(* Logix 5000 project; controller PLCbox vendor 1 type 14 code 149 rev 30.11; software revision 30.01; part 4 of 4 *)
(* tags used below, declared in another part *)
   AScaled : REAL;
   BOOL : BOOL[64];
   LocalBOOL : BOOL[64];
   LocalDINT : DINT[20];
   LocDINT : DINT[20];
   MTR1 : BOOL[64];
   Running : BOOL;
   StartPB : BOOL;
   StopButton : BOOL;
   StopPB : DINT;
   TempC : REAL;
   TempF : REAL;
   AnalogInput : REAL[100];
   DINT_Arr1 : DINT[40];
   DINT_Arr2 : DINT[40];
   FaultedT : TIMER;
   HMI_Int_BOOL : BOOL[64];
   Light1_Complete_ONS : BOOL;
   Light1_Green : BOOL;
   Light1_Green_T : TIMER;
   Light1_Red : BOOL;
   Light1_Reset : BOOL;
   Light1_Yellow : BOOL;
   Light1_Yellow_T : TIMER;
   Light2_Complete_ONS : BOOL;
   Light2_Green : BOOL;
   Light2_Green_T : TIMER;
   Light2_Red : BOOL;
   Light2_Reset : BOOL;
   Light2_Yellow : BOOL;
   Light2_Yellow_T : TIMER;
   LightSystem_FLT : BOOL[64];
   LightSystemFaulted : BOOL;
   Local2IData : DINT;
   Local3OData : DINT;
   Local_IN_D : BOOL[256];
   Local_OUT_D : BOOL[256];
   System_Timer : TIMER[100];
   SystemFaultReset : BOOL;
   tagToPi : DINT;
(* ST_Practice, continued *)

ROUTINE _04_MotorStartST   (* structured text *)
   // MTR1[3] - StartPB
   // MTR1[4] - StopPB
   // MTR1[5] - Motor Running
   //MTR1[5] := (MTR1[3] OR MTR1[5]) AND NOT(MTR1[4]);
   IF (MTR1[3] OR MTR1[5]) AND NOT(MTR1[4]) THEN
   MTR1[5] := 1;
   ELSE
   MTR1[5] := 0;
   END_IF;
END_ROUTINE

ROUTINE _05_Practice   (* structured text *)
   
END_ROUTINE

ROUTINE _06_LogicOps   (* structured text *)
   //OR Operator
   LocalBOOL[0] := LocalBOOL[1] OR LocalBOOL[2];
   
   //AND Operator
   LocalBOOL[3] := LocalBOOL[4] AND LocalBOOL[5];
   
   //NOT Operator
   LocalBOOL[6] := NOT(LocalBOOL[7]);
   
   //Motor Starter
   Running [:=] (Running OR StartPB) AND NOT(StopButton);
   
   //GRT, LES, LIM (Not available in ST) -> CMP
   LocalBOOL[8] := 100 + LocalDINT[1] < LocalDINT[0] - 44;
END_ROUTINE

ROUTINE _07_OperatorsFunctions   (* structured text *)
   //Mathematical / Built-In Operators
   LocDINT[0] := LocDINT[1] + 5;
   LocDINT[2] := LocDINT[3] - 4;
   LocDINT[4] := LocDINT[0] * 3;
   LocDINT[5] := 5/LocDINT[1];
   LocDINT[6] := LocDINT[0] ** 3;
   LocDINT[7] := LocDINT[6] MOD 4;
   
   LocDINT[8] := LocDINT[1] + LocDINT[6] / 2 + LocDINT[2];
   
   //Examples
   TempC := (TempF - 32) * 5/9;
   AScaled := AnalogInput[0] / 160 * 3;
END_ROUTINE
END_PROGRAM

PROGRAM StreetLightSystem   (* main routine _01_Main *)
VAR
   HMI_Int_DINT : DINT[100] := ([0] := 10000, [1] := 3000, [2] := 10000, [3] := 3000);
END_VAR

ROUTINE _01_Main   (* ladder *)
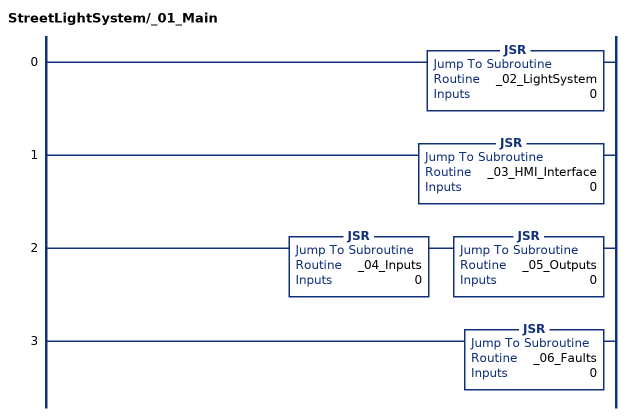
   0: JSR(_02_LightSystem,0);
   1: JSR(_03_HMI_Interface,0);
   2: JSR(_04_Inputs,0)JSR(_05_Outputs,0);
   3: JSR(_06_Faults,0);
END_ROUTINE

ROUTINE _02_LightSystem   (* ladder *)
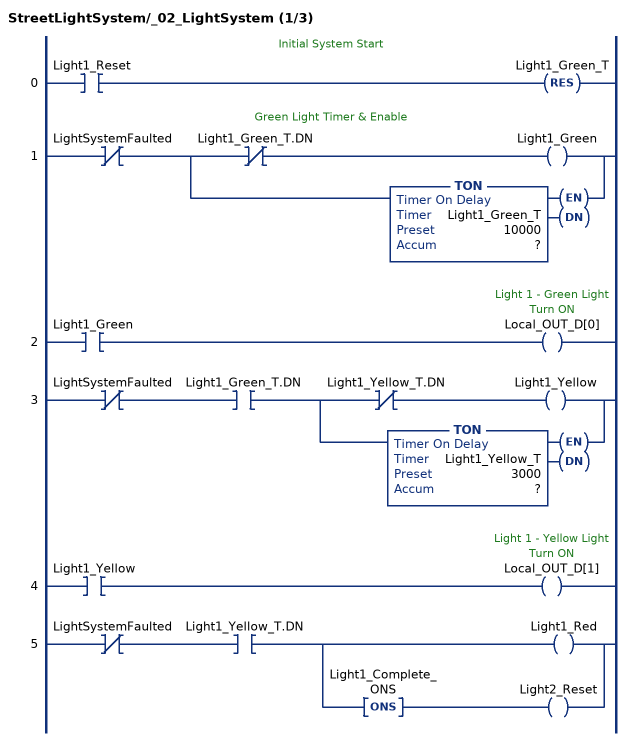
   // Initial System Start
   0: XIC(Light1_Reset)RES(Light1_Green_T);
   // Green Light Timer & Enable
   1: XIO(LightSystemFaulted)[XIO(Light1_Green_T.DN) OTE(Light1_Green) ,TON(Light1_Green_T,?,?) ];
   2: XIC(Light1_Green)OTE(Local_OUT_D[0]);
   3: XIO(LightSystemFaulted)XIC(Light1_Green_T.DN)[XIO(Light1_Yellow_T.DN) OTE(Light1_Yellow) ,TON(Light1_Yellow_T,?,?) ];
   4: XIC(Light1_Yellow)OTE(Local_OUT_D[1]);
   5: XIO(LightSystemFaulted)XIC(Light1_Yellow_T.DN)[OTE(Light1_Red) ,ONS(Light1_Complete_ONS) OTE(Light2_Reset) ];
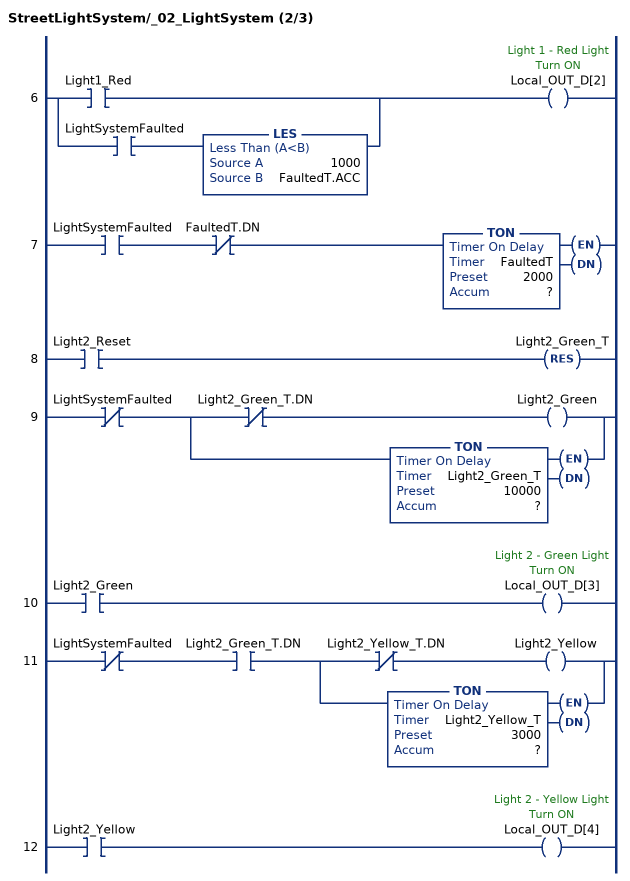
   6: [XIC(Light1_Red) ,XIC(LightSystemFaulted) LES(1000,FaultedT.ACC) ]OTE(Local_OUT_D[2]);
   7: XIC(LightSystemFaulted)XIO(FaultedT.DN)TON(FaultedT,?,?);
   8: XIC(Light2_Reset)RES(Light2_Green_T);
   9: XIO(LightSystemFaulted)[XIO(Light2_Green_T.DN) OTE(Light2_Green) ,TON(Light2_Green_T,?,?) ];
   10: XIC(Light2_Green)OTE(Local_OUT_D[3]);
   11: XIO(LightSystemFaulted)XIC(Light2_Green_T.DN)[XIO(Light2_Yellow_T.DN) OTE(Light2_Yellow) ,TON(Light2_Yellow_T,?,?) ];
   12: XIC(Light2_Yellow)OTE(Local_OUT_D[4]);
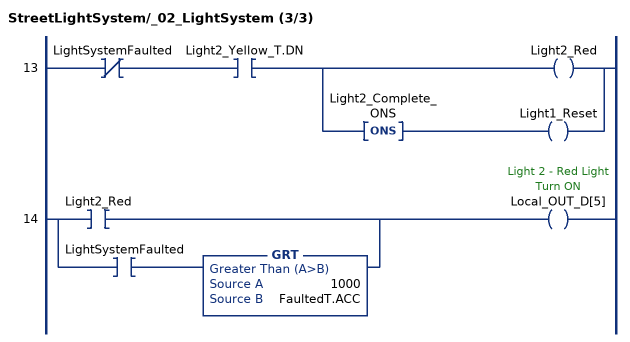
   13: XIO(LightSystemFaulted)XIC(Light2_Yellow_T.DN)[OTE(Light2_Red) ,ONS(Light2_Complete_ONS) OTE(Light1_Reset) ];
   14: [XIC(Light2_Red) ,XIC(LightSystemFaulted) GRT(1000,FaultedT.ACC) ]OTE(Local_OUT_D[5]);
END_ROUTINE

ROUTINE _03_HMI_Interface   (* ladder *)
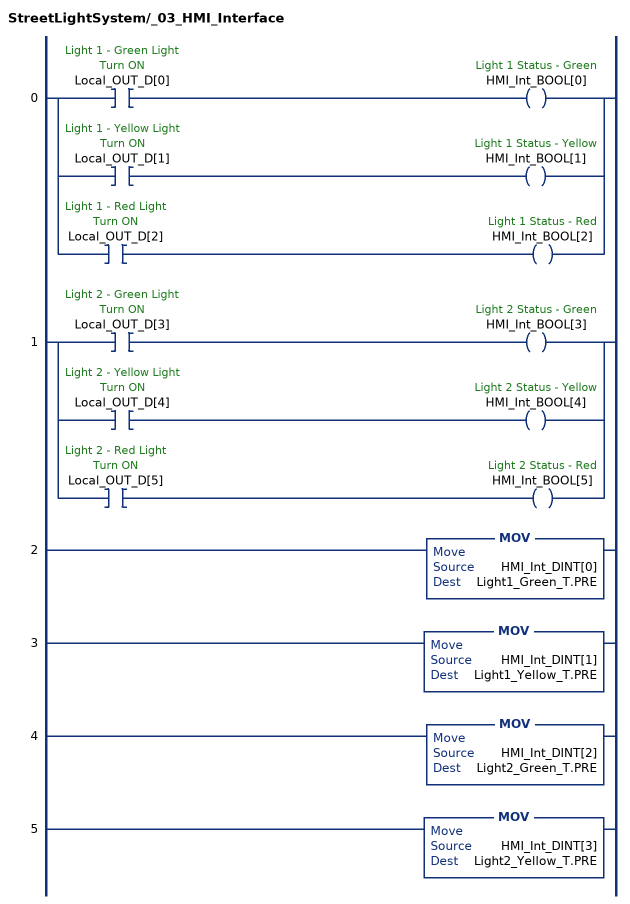
   0: [XIC(Local_OUT_D[0]) OTE(HMI_Int_BOOL[0]) ,XIC(Local_OUT_D[1]) OTE(HMI_Int_BOOL[1]) ,XIC(Local_OUT_D[2]) OTE(HMI_Int_BOOL[2]) ];
   1: [XIC(Local_OUT_D[3]) OTE(HMI_Int_BOOL[3]) ,XIC(Local_OUT_D[4]) OTE(HMI_Int_BOOL[4]) ,XIC(Local_OUT_D[5]) OTE(HMI_Int_BOOL[5]) ];
   2: MOV(HMI_Int_DINT[0],Light1_Green_T.PRE);
   3: MOV(HMI_Int_DINT[1],Light1_Yellow_T.PRE);
   4: MOV(HMI_Int_DINT[2],Light2_Green_T.PRE);
   5: MOV(HMI_Int_DINT[3],Light2_Yellow_T.PRE);
END_ROUTINE

ROUTINE _04_Inputs   (* ladder *)
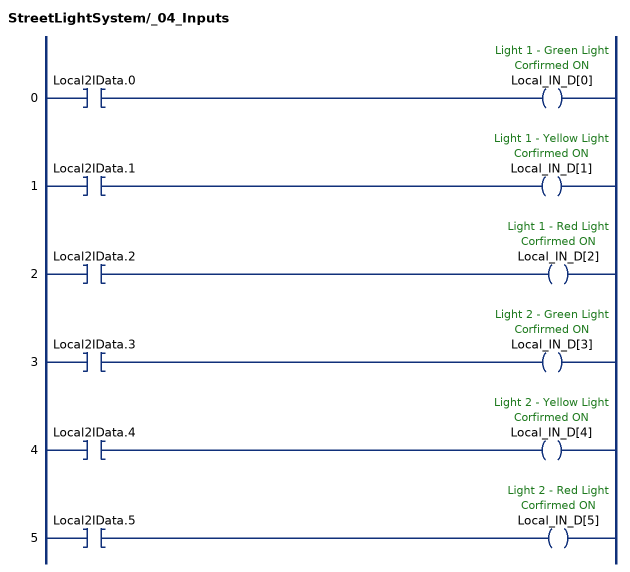
   0: XIC(Local2IData.0)OTE(Local_IN_D[0]);
   1: XIC(Local2IData.1)OTE(Local_IN_D[1]);
   2: XIC(Local2IData.2)OTE(Local_IN_D[2]);
   3: XIC(Local2IData.3)OTE(Local_IN_D[3]);
   4: XIC(Local2IData.4)OTE(Local_IN_D[4]);
   5: XIC(Local2IData.5)OTE(Local_IN_D[5]);
END_ROUTINE

ROUTINE _05_Outputs   (* ladder *)
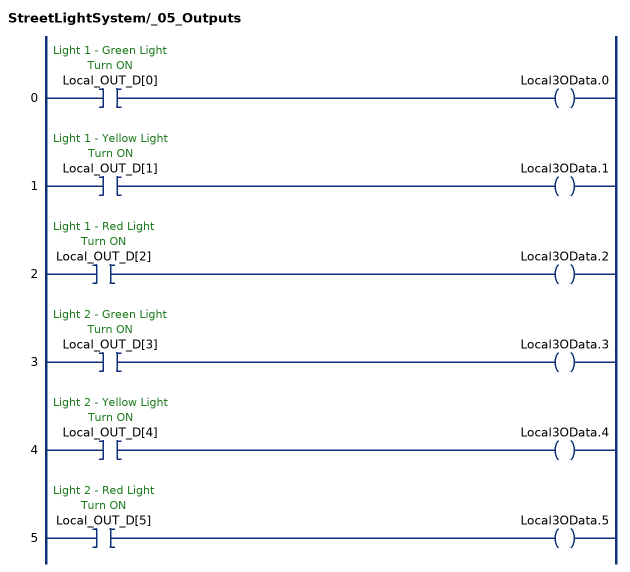
   0: XIC(Local_OUT_D[0])OTE(Local3OData.0);
   1: XIC(Local_OUT_D[1])OTE(Local3OData.1);
   2: XIC(Local_OUT_D[2])OTE(Local3OData.2);
   3: XIC(Local_OUT_D[3])OTE(Local3OData.3);
   4: XIC(Local_OUT_D[4])OTE(Local3OData.4);
   5: XIC(Local_OUT_D[5])OTE(Local3OData.5);
END_ROUTINE

ROUTINE _06_Faults   (* ladder *)
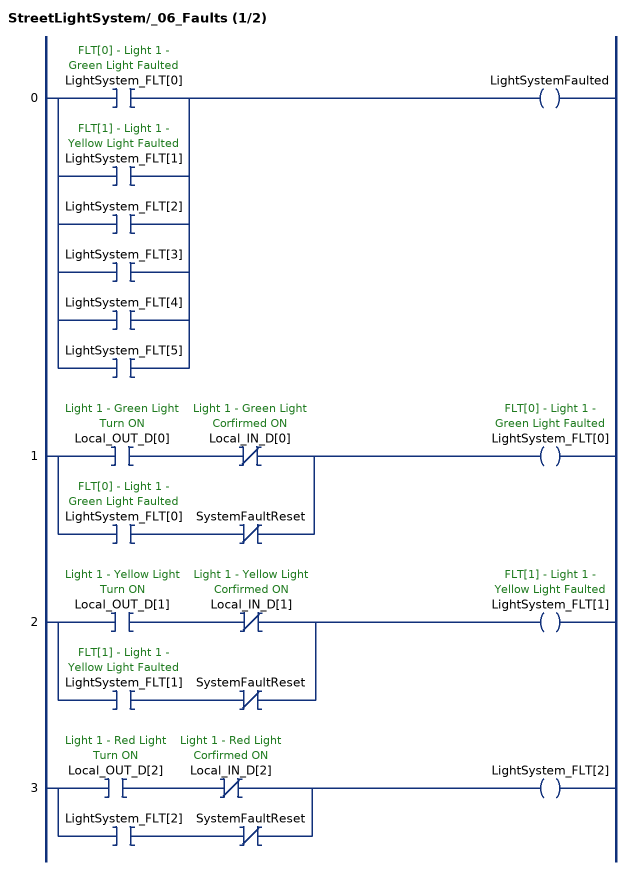
   0: [XIC(LightSystem_FLT[0]) ,XIC(LightSystem_FLT[1]) ,XIC(LightSystem_FLT[2]) ,XIC(LightSystem_FLT[3]) ,XIC(LightSystem_FLT[4]) ,XIC(LightSystem_FLT[5]) ]OTE(LightSystemFaulted);
   1: [XIC(Local_OUT_D[0]) XIO(Local_IN_D[0]) ,XIC(LightSystem_FLT[0]) XIO(SystemFaultReset) ]OTE(LightSystem_FLT[0]);
   2: [XIC(Local_OUT_D[1]) XIO(Local_IN_D[1]) ,XIC(LightSystem_FLT[1]) XIO(SystemFaultReset) ]OTE(LightSystem_FLT[1]);
   3: [XIC(Local_OUT_D[2]) XIO(Local_IN_D[2]) ,XIC(LightSystem_FLT[2]) XIO(SystemFaultReset) ]OTE(LightSystem_FLT[2]);
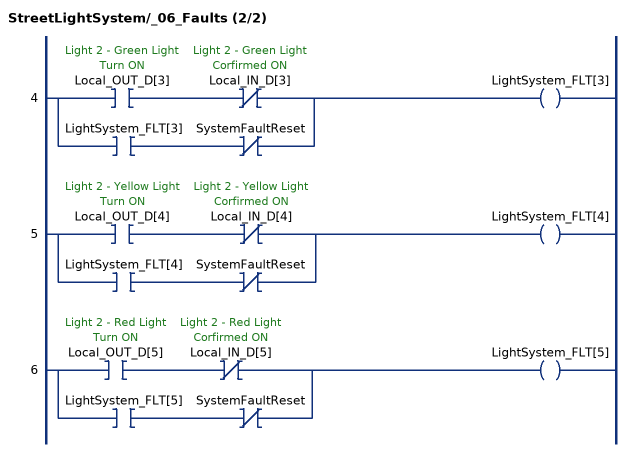
   4: [XIC(Local_OUT_D[3]) XIO(Local_IN_D[3]) ,XIC(LightSystem_FLT[3]) XIO(SystemFaultReset) ]OTE(LightSystem_FLT[3]);
   5: [XIC(Local_OUT_D[4]) XIO(Local_IN_D[4]) ,XIC(LightSystem_FLT[4]) XIO(SystemFaultReset) ]OTE(LightSystem_FLT[4]);
   6: [XIC(Local_OUT_D[5]) XIO(Local_IN_D[5]) ,XIC(LightSystem_FLT[5]) XIO(SystemFaultReset) ]OTE(LightSystem_FLT[5]);
END_ROUTINE
END_PROGRAM

PROGRAM TankFillingChallenge   (* main routine _01_Main *)
VAR
   DischargeStatus : DINT := 1;
   FillingStatus : DINT := 1;
   T_Vlad : BOOL[128];
   TankActualLevel : REAL := 42.792046;
   TankDischargeRate : REAL := 0.5;
   TankEmptyThreshold : REAL := 5.0;
   TankFill : BOOL[128];
        [6]   // TANK FULL
        [7]   // TANK EMPTY
        [2]   // Filling Station RUNNING
        [3]   // START Discharge Station
        [0]   // START Filling Station
        [1]   // STOP Filling Station
        [5]   // Discharge Station RUNNING
        [4]   // STOP Discharge Station
   TankFillRate : REAL := 0.3;
   TankFullThreshold : REAL := 100.0;
   TankOut : BOOL[32];
        [0]   // Filling Station VALVE OPEN
        [1]   // Discharge Station VALVE OPEN
   TankTimers : TIMER[10] := ([0].PRE := 20, [1].PRE := 20);
END_VAR

ROUTINE _01_Main   (* ladder *)
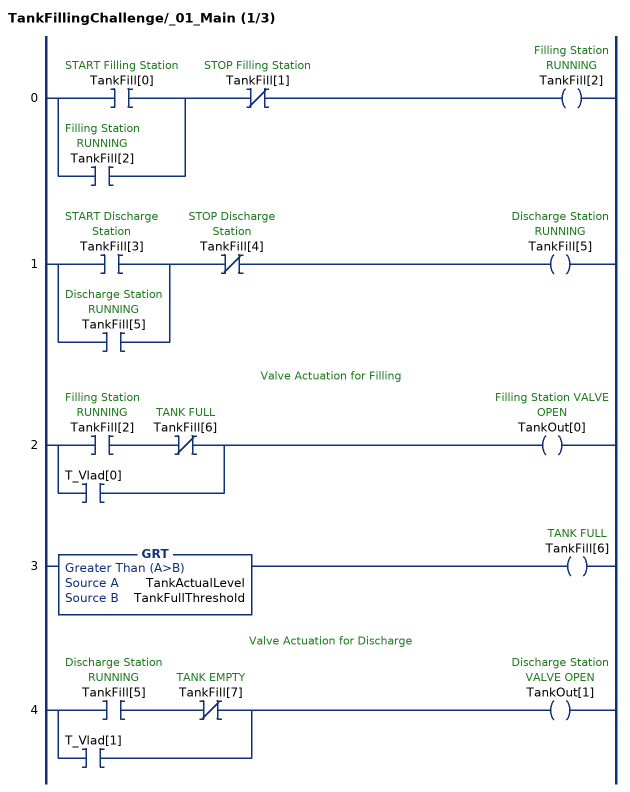
   0: [XIC(TankFill[0]) ,XIC(TankFill[2]) ]XIO(TankFill[1])OTE(TankFill[2]);
   1: [XIC(TankFill[3]) ,XIC(TankFill[5]) ]XIO(TankFill[4])OTE(TankFill[5]);
   // Valve Actuation for Filling
   2: [XIC(TankFill[2]) XIO(TankFill[6]) ,XIC(T_Vlad[0]) ]OTE(TankOut[0]);
   3: GRT(TankActualLevel,TankFullThreshold)OTE(TankFill[6]);
   // Valve Actuation for Discharge
   4: [XIC(TankFill[5]) XIO(TankFill[7]) ,XIC(T_Vlad[1]) ]OTE(TankOut[1]);
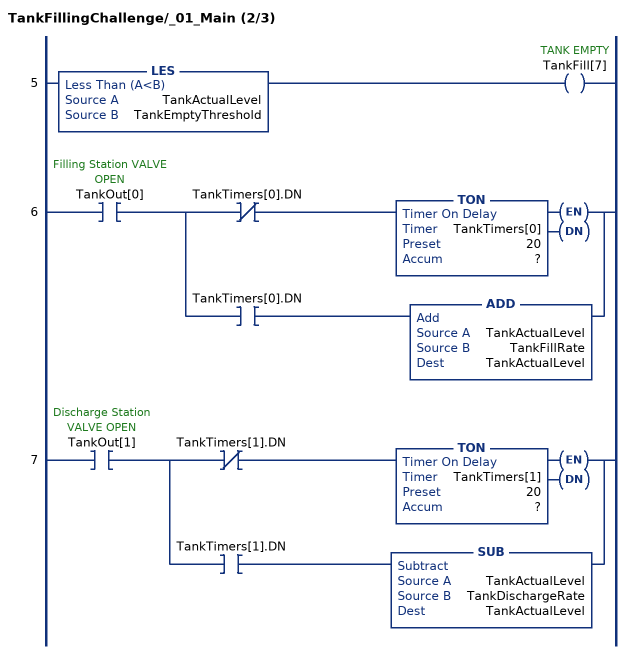
   5: LES(TankActualLevel,TankEmptyThreshold)OTE(TankFill[7]);
   6: XIC(TankOut[0])[XIO(TankTimers[0].DN) TON(TankTimers[0],?,?) ,XIC(TankTimers[0].DN) ADD(TankActualLevel,TankFillRate,TankActualLevel) ];
   7: XIC(TankOut[1])[XIO(TankTimers[1].DN) TON(TankTimers[1],?,?) ,XIC(TankTimers[1].DN) SUB(TankActualLevel,TankDischargeRate,TankActualLevel) ];
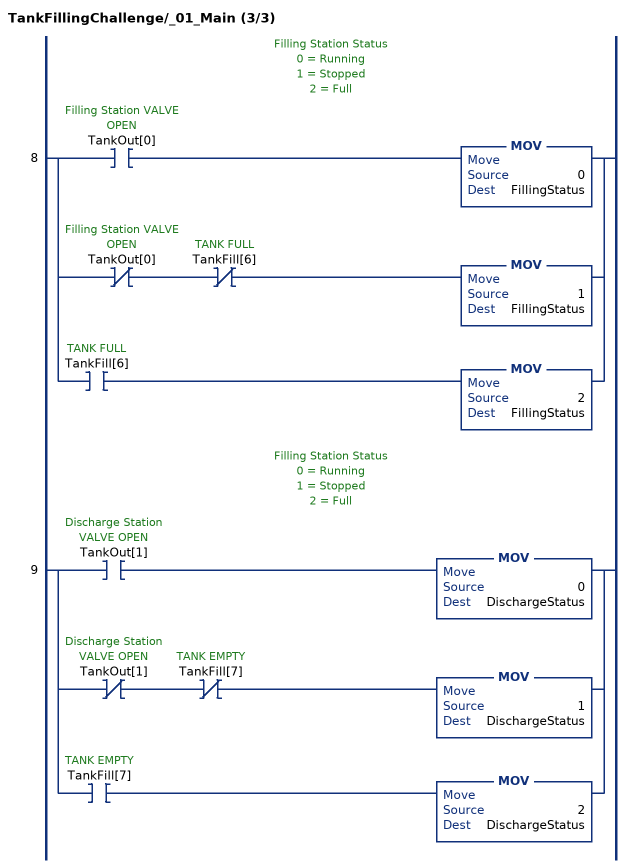
   // Filling Station Status
   // 0 = Running
   // 1 = Stopped
   // 2 = Full
   8: [XIC(TankOut[0]) MOV(0,FillingStatus) ,XIO(TankOut[0]) XIO(TankFill[6]) MOV(1,FillingStatus) ,XIC(TankFill[6]) MOV(2,FillingStatus) ];
   // Filling Station Status
   // 0 = Running
   // 1 = Stopped
   // 2 = Full
   9: [XIC(TankOut[1]) MOV(0,DischargeStatus) ,XIO(TankOut[1]) XIO(TankFill[7]) MOV(1,DischargeStatus) ,XIC(TankFill[7]) MOV(2,DischargeStatus) ];
END_ROUTINE
END_PROGRAM

PROGRAM TestProgram   (* main routine Main *)
VAR
   ALARM : BOOL[256];
   ALARM2 : BOOL[256];
   ALARM_DESC : String20;
   ALARM_DESCR : String20[256] := ([0] := 'Fault 0', [1] := 'Fault 1', [2] := 'Fault 2');
   Condition1 : BOOL := 1;
   Condition10 : BOOL := 1;
   Condition11 : BOOL := 1;
   Condition2 : BOOL;
   Condition3 : BOOL := 1;
   Condition4 : BOOL;
   Condition5 : BOOL := 1;
   Condition6 : BOOL;
   Condition7 : BOOL;
   Condition8 : BOOL := 1;
   Condition9 : BOOL := 1;
   EmptyString : String20;
   Energize : BOOL;
   Energize1 : BOOL := 1;
   FaultDesc : String20 := 'Fault 1';
   FaultDesc2 : String20 := 'Fault 1';
   HMI_BOOL : BOOL[32];
   Index : DINT := 256;
   Motor_1_Start : BOOL;
   Motor_2_Start : BOOL;
   OFFinst : TIMER := (PRE := 500);
   ONinst : TIMER := (PRE := 3000, ACC := 2342, EN := 1, TT := 1);
   PLC_BOOL : BOOL[32];
   Program_Enabled : BOOL;
   Program_Running : BOOL;
   Program_Starting : BOOL;
   RunRoutine : TIMER := (PRE := 500);
   StartProgram : BOOL;
   StartRoutine : TIMER := (PRE := 1000);
   System_Cond : BOOL[256] := ([0] := 1);
        [0]   // Start MOTOR 1
        [2]   // Start MOTOR 2
        [5]   // Boiler at Temp
        [6]   // System Running
        [7]   // System FAULTED
        [1]   // MOTOR 1 At Target Speed
        [8]   // System RESET
        [4]   // Heat Boiler
        [3]   // Motor 2 at Target Speed
   System_INT : INT[10] := ([0] := 456, [1] := 456, [2] := 1);
   System_REAL : REAL[10] := ([0] := 54.0, [1] := 54.0, [2] := 54.0);
   System_STR : STRING[10];
   System_STRING : String20[10];
   SystemFaulted : BOOL := 1;
   SystemFaulted2 : BOOL := 1;
   SystemStart : BOOL;
   SytemReset : BOOL;
   SytemReset2 : BOOL;
   Test1 : DINT := 560647;
   Test2 : INT := -29177;
   TestDINT : DINT;
   TestINT : INT;
END_VAR

ROUTINE _02_MOV_Instruction   (* ladder *)
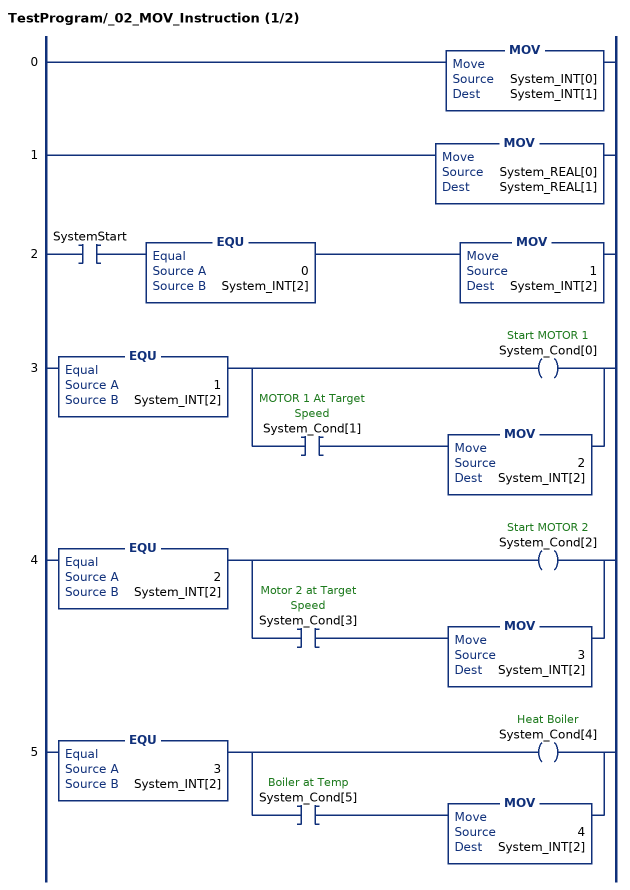
   0: MOV(System_INT[0],System_INT[1]);
   1: MOV(System_REAL[0],System_REAL[1]);
   2: XIC(SystemStart)EQU(0,System_INT[2])MOV(1,System_INT[2]);
   3: EQU(1,System_INT[2])[OTE(System_Cond[0]) ,XIC(System_Cond[1]) MOV(2,System_INT[2]) ];
   4: EQU(2,System_INT[2])[OTE(System_Cond[2]) ,XIC(System_Cond[3]) MOV(3,System_INT[2]) ];
   5: EQU(3,System_INT[2])[OTE(System_Cond[4]) ,XIC(System_Cond[5]) MOV(4,System_INT[2]) ];
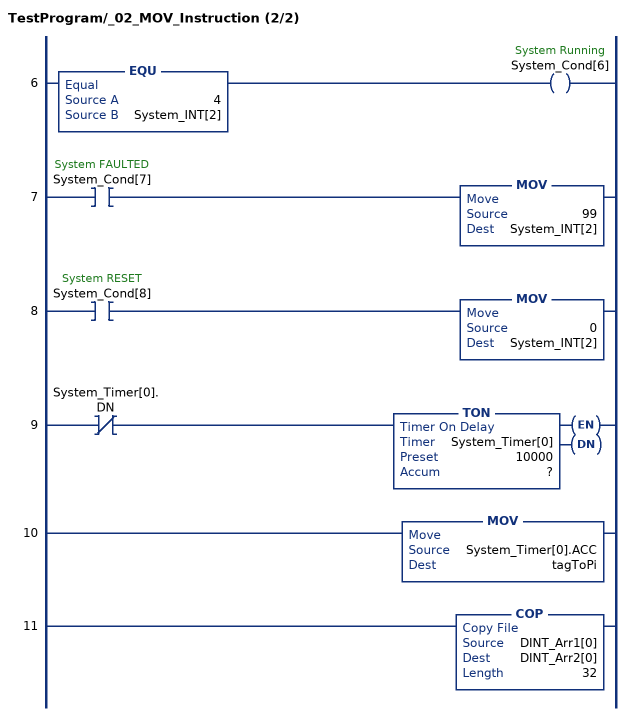
   6: EQU(4,System_INT[2])OTE(System_Cond[6]);
   7: XIC(System_Cond[7])MOV(99,System_INT[2]);
   8: XIC(System_Cond[8])MOV(0,System_INT[2]);
   9: XIO(System_Timer[0].DN)TON(System_Timer[0],?,?);
   10: MOV(System_Timer[0].ACC,tagToPi);
   11: COP(DINT_Arr1[0],DINT_Arr2[0],32);
END_ROUTINE

ROUTINE _03_HMI   (* ladder *)
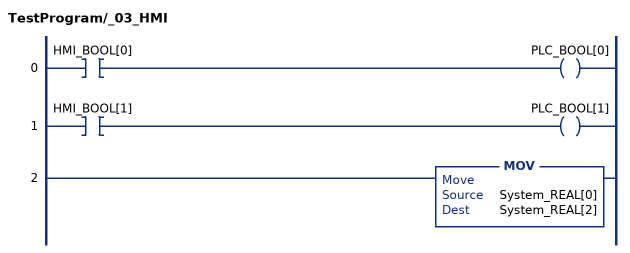
   0: XIC(HMI_BOOL[0])OTE(PLC_BOOL[0]);
   1: XIC(HMI_BOOL[1])OTE(PLC_BOOL[1]);
   2: MOV(System_REAL[0],System_REAL[2]);
END_ROUTINE

ROUTINE _04_Ladder   (* ladder *)
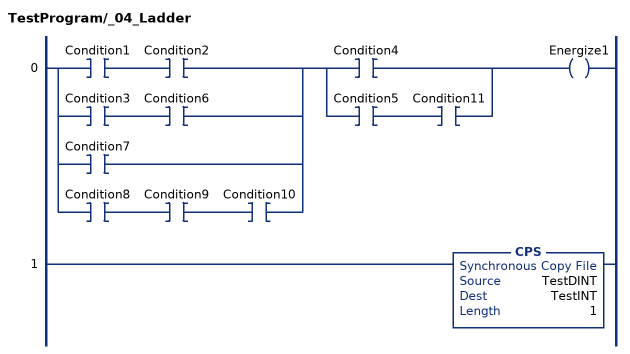
   0: [XIC(Condition1) XIC(Condition2) ,[XIC(Condition3) XIC(Condition6) ,XIC(Condition7) ] ,XIC(Condition8) XIC(Condition9) XIC(Condition10) ][XIC(Condition4) ,XIC(Condition5) XIC(Condition11) ]OTE(Energize1);
   1: CPS(TestDINT,TestINT,1);
END_ROUTINE

ROUTINE Main   (* ladder *)
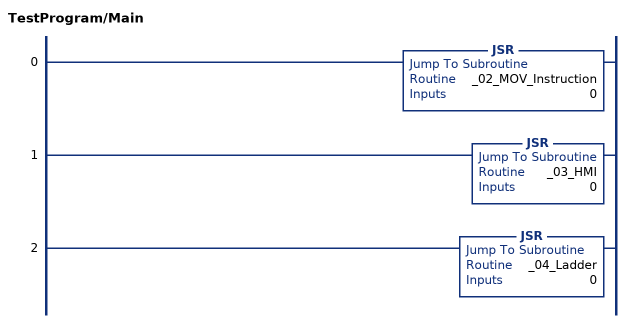
   0: JSR(_02_MOV_Instruction,0);
   1: JSR(_03_HMI,0);
   2: JSR(_04_Ladder,0);
END_ROUTINE
END_PROGRAM
